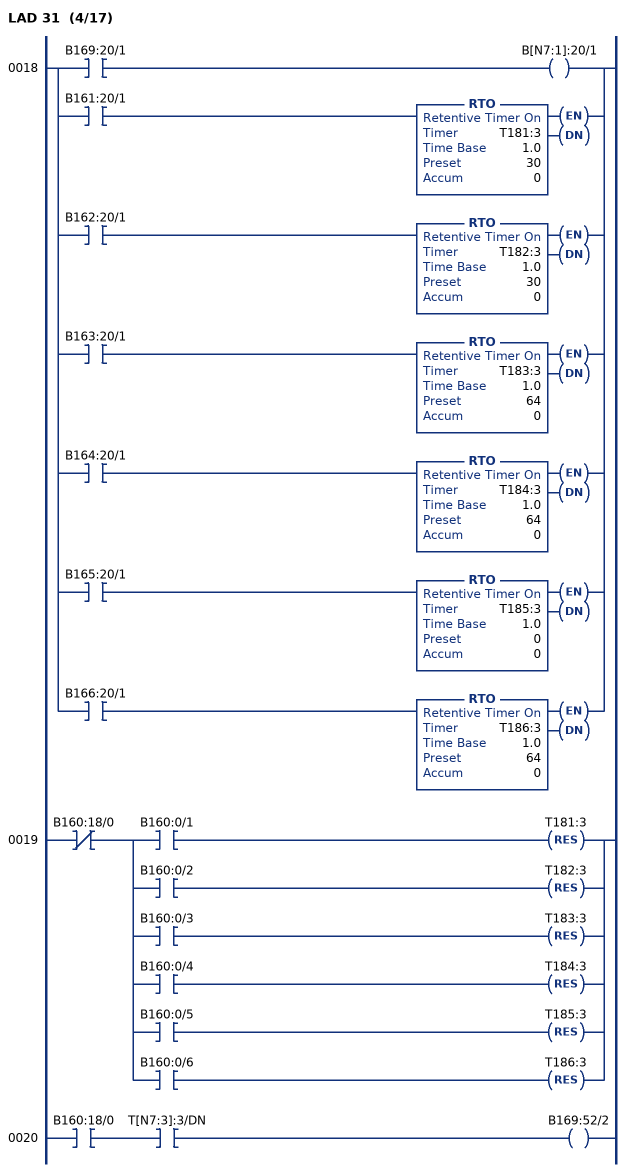
% Rung: 18 %
SOR BST XIC B169:20/1 OTE B[N7:1]:20/1 NXB XIC B161:20/1 RTO T181:3 1.0 30 0 NXB XIC B162:20/1 RTO T182:3 1.0 30 0 NXB XIC B163:20/1 RTO T183:3 1.0 64 0 NXB XIC B164:20/1 RTO T184:3 1.0 64 0 NXB XIC B165:20/1 RTO T185:3 1.0 0 0 NXB XIC B166:20/1 RTO T186:3 1.0 64 0 BND EOR
% Rung: 19 %
SOR XIO B160:18/0 BST XIC B160:0/1 RES T181:3 NXB XIC B160:0/2 RES T182:3 NXB XIC B160:0/3 RES T183:3 NXB XIC B160:0/4 RES T184:3 NXB XIC B160:0/5 RES T185:3 NXB XIC B160:0/6 RES T186:3 BND EOR
% Rung: 20 %
SOR XIC B160:18/0 XIC T[N7:3]:3/DN OTE B169:52/2 EOR

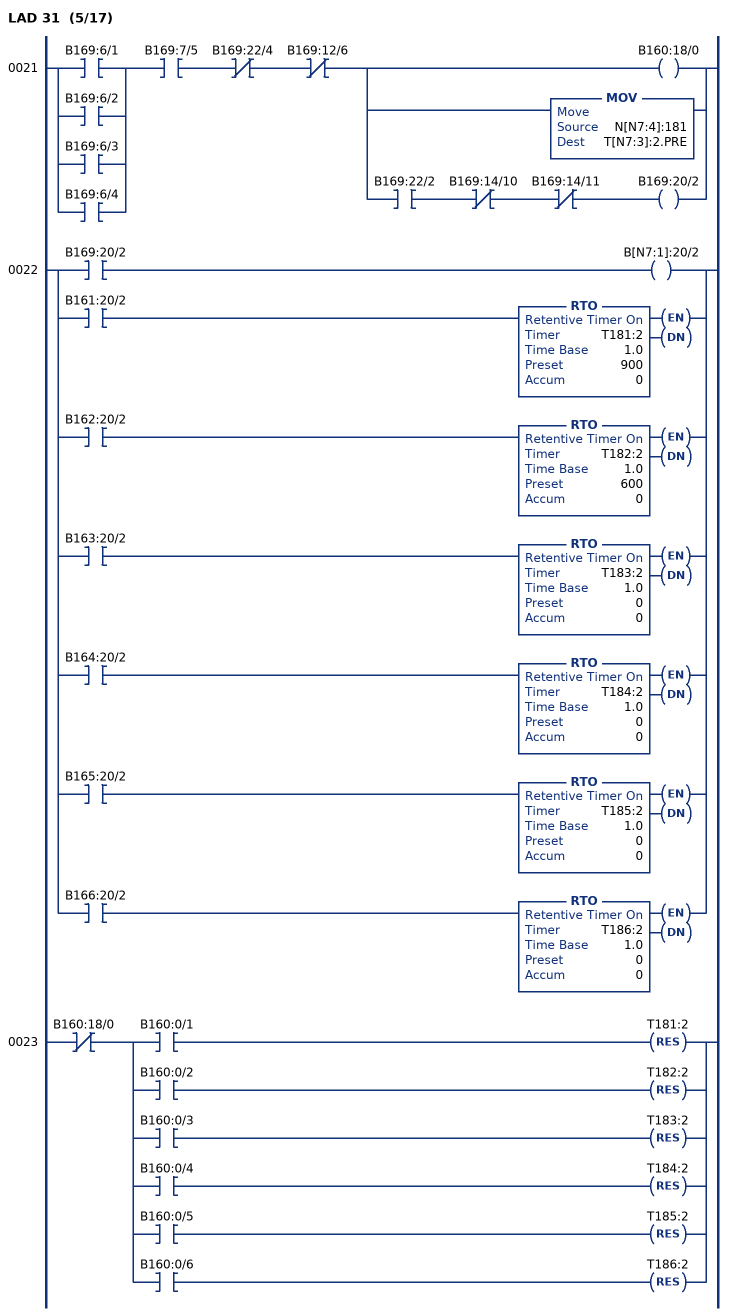
% Rung: 21 %
SOR BST XIC B169:6/1 NXB XIC B169:6/2 NXB XIC B169:6/3 NXB XIC B169:6/4 BND XIC B169:7/5 XIO B169:22/4 XIO B169:12/6 BST OTE B160:18/0 NXB MOV N[N7:4]:181 T[N7:3]:2.PRE NXB XIC B169:22/2 XIO B169:14/10 XIO B169:14/11 OTE B169:20/2 BND EOR
% Rung: 22 %
SOR BST XIC B169:20/2 OTE B[N7:1]:20/2 NXB XIC B161:20/2 RTO T181:2 1.0 900 0 NXB XIC B162:20/2 RTO T182:2 1.0 600 0 NXB XIC B163:20/2 RTO T183:2 1.0 0 0 NXB XIC B164:20/2 RTO T184:2 1.0 0 0 NXB XIC B165:20/2 RTO T185:2 1.0 0 0 NXB XIC B166:20/2 RTO T186:2 1.0 0 0 BND EOR
% Rung: 23 %
SOR XIO B160:18/0 BST XIC B160:0/1 RES T181:2 NXB XIC B160:0/2 RES T182:2 NXB XIC B160:0/3 RES T183:2 NXB XIC B160:0/4 RES T184:2 NXB XIC B160:0/5 RES T185:2 NXB XIC B160:0/6 RES T186:2 BND EOR

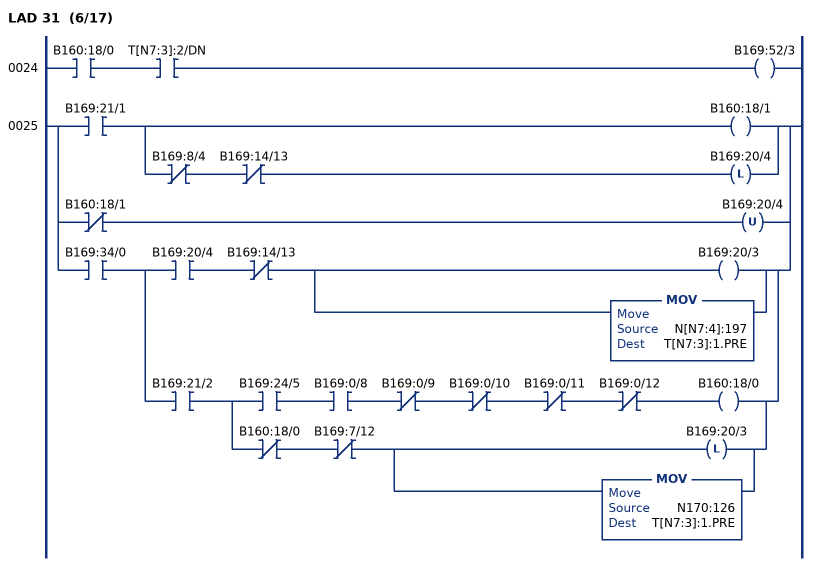
% Rung: 24 %
SOR XIC B160:18/0 XIC T[N7:3]:2/DN OTE B169:52/3 EOR
% Rung: 25 %
SOR BST XIC B169:21/1 BST OTE B160:18/1 NXB XIO B169:8/4 XIO B169:14/13 OTL B169:20/4 BND NXB XIO B160:18/1 OTU B169:20/4 NXB XIC B169:34/0 BST XIC B169:20/4 XIO B169:14/13 BST OTE B169:20/3 NXB MOV N[N7:4]:197 T[N7:3]:1.PRE BND NXB XIC B169:21/2 BST XIC B169:24/5 XIC B169:0/8 XIO B169:0/9 XIO B169:0/10 XIO B169:0/11 XIO B169:0/12 OTE B160:18/0 NXB XIO B160:18/0 XIO B169:7/12 BST OTL B169:20/3 NXB MOV N170:126 T[N7:3]:1.PRE BND BND BND BND EOR

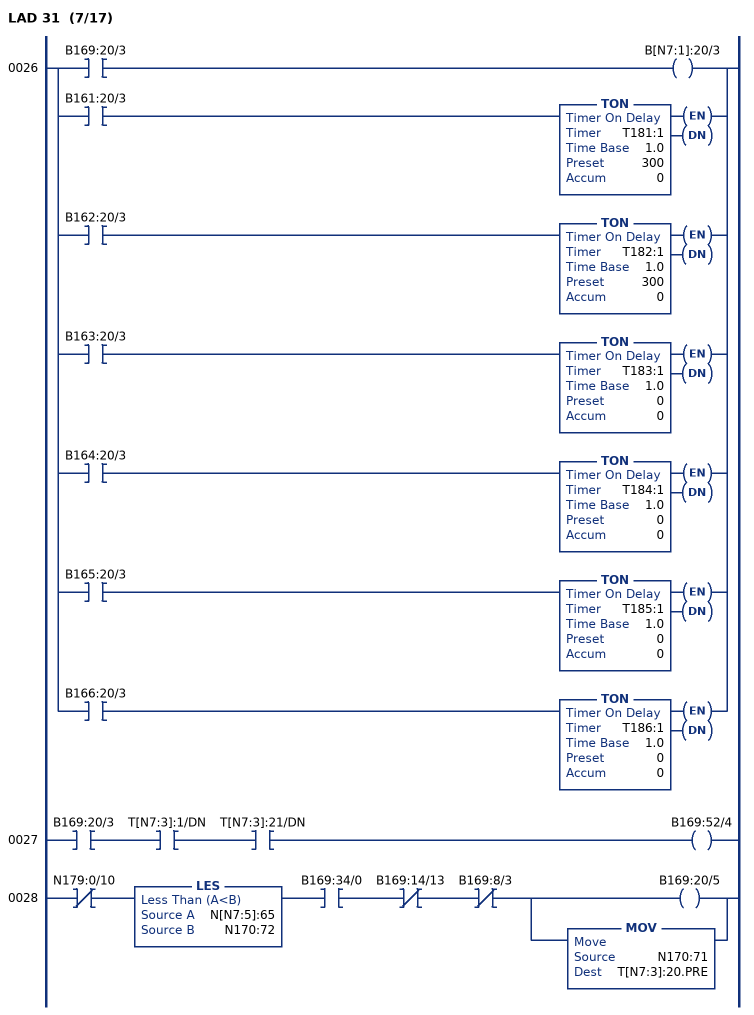
% Rung: 26 %
SOR BST XIC B169:20/3 OTE B[N7:1]:20/3 NXB XIC B161:20/3 TON T181:1 1.0 300 0 NXB XIC B162:20/3 TON T182:1 1.0 300 0 NXB XIC B163:20/3 TON T183:1 1.0 0 0 NXB XIC B164:20/3 TON T184:1 1.0 0 0 NXB XIC B165:20/3 TON T185:1 1.0 0 0 NXB XIC B166:20/3 TON T186:1 1.0 0 0 BND EOR
% Rung: 27 %
SOR XIC B169:20/3 XIC T[N7:3]:1/DN XIC T[N7:3]:21/DN OTE B169:52/4 EOR
% Rung: 28 %
SOR XIO N179:0/10 LES N[N7:5]:65 N170:72 XIC B169:34/0 XIO B169:14/13 XIO B169:8/3 BST OTE B169:20/5 NXB MOV N170:71 T[N7:3]:20.PRE BND EOR

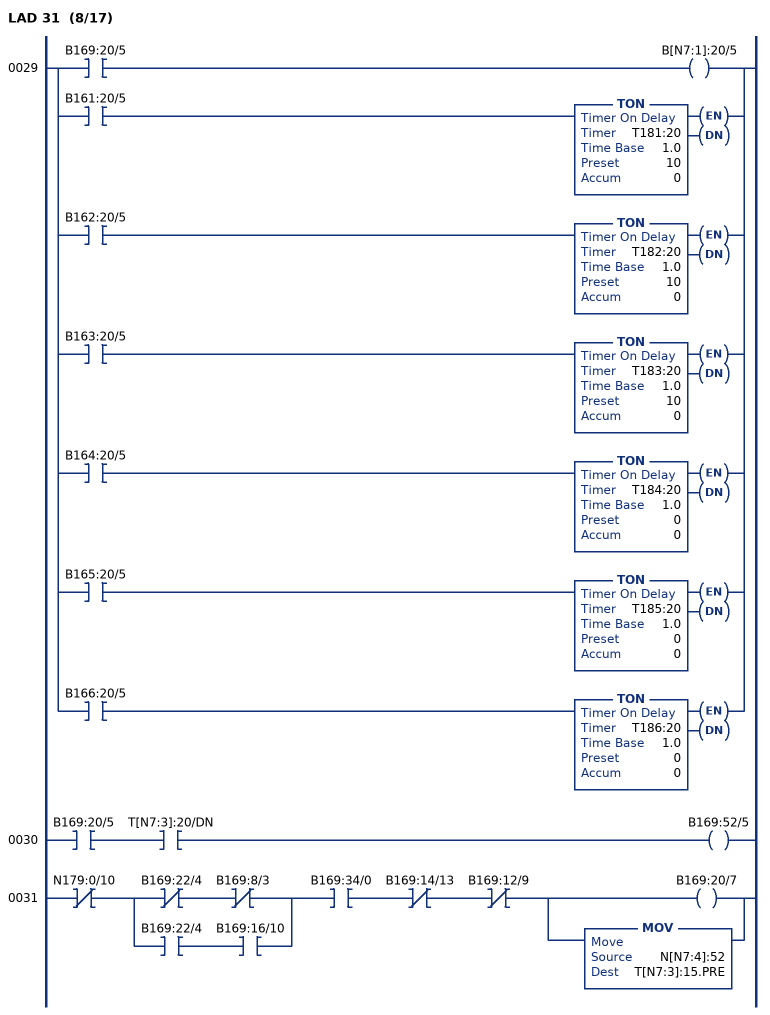
% Rung: 29 %
SOR BST XIC B169:20/5 OTE B[N7:1]:20/5 NXB XIC B161:20/5 TON T181:20 1.0 10 0 NXB XIC B162:20/5 TON T182:20 1.0 10 0 NXB XIC B163:20/5 TON T183:20 1.0 10 0 NXB XIC B164:20/5 TON T184:20 1.0 0 0 NXB XIC B165:20/5 TON T185:20 1.0 0 0 NXB XIC B166:20/5 TON T186:20 1.0 0 0 BND EOR
% Rung: 30 %
SOR XIC B169:20/5 XIC T[N7:3]:20/DN OTE B169:52/5 EOR
% Rung: 31 %
SOR XIO N179:0/10 BST XIO B169:22/4 XIO B169:8/3 NXB XIC B169:22/4 XIC B169:16/10 BND XIC B169:34/0 XIO B169:14/13 XIO B169:12/9 BST OTE B169:20/7 NXB MOV N[N7:4]:52 T[N7:3]:15.PRE BND EOR

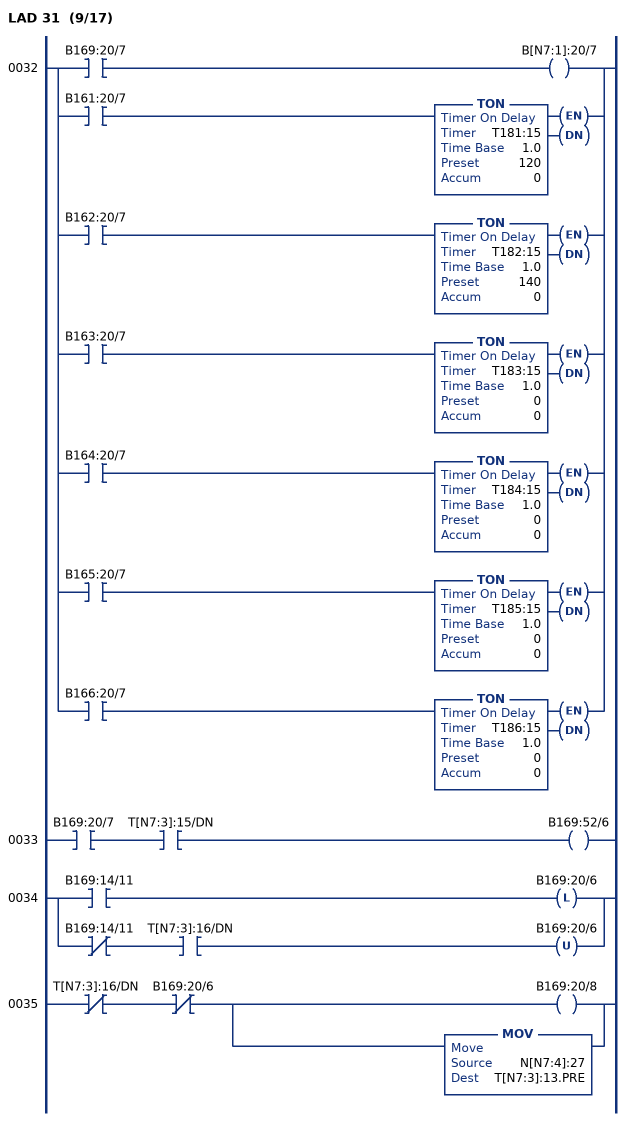
% Rung: 32 %
SOR BST XIC B169:20/7 OTE B[N7:1]:20/7 NXB XIC B161:20/7 TON T181:15 1.0 120 0 NXB XIC B162:20/7 TON T182:15 1.0 140 0 NXB XIC B163:20/7 TON T183:15 1.0 0 0 NXB XIC B164:20/7 TON T184:15 1.0 0 0 NXB XIC B165:20/7 TON T185:15 1.0 0 0 NXB XIC B166:20/7 TON T186:15 1.0 0 0 BND EOR
% Rung: 33 %
SOR XIC B169:20/7 XIC T[N7:3]:15/DN OTE B169:52/6 EOR
% Rung: 34 %
SOR BST XIC B169:14/11 OTL B169:20/6 NXB XIO B169:14/11 XIC T[N7:3]:16/DN OTU B169:20/6 BND EOR
% Rung: 35 %
SOR XIO T[N7:3]:16/DN XIO B169:20/6 BST OTE B169:20/8 NXB MOV N[N7:4]:27 T[N7:3]:13.PRE BND EOR

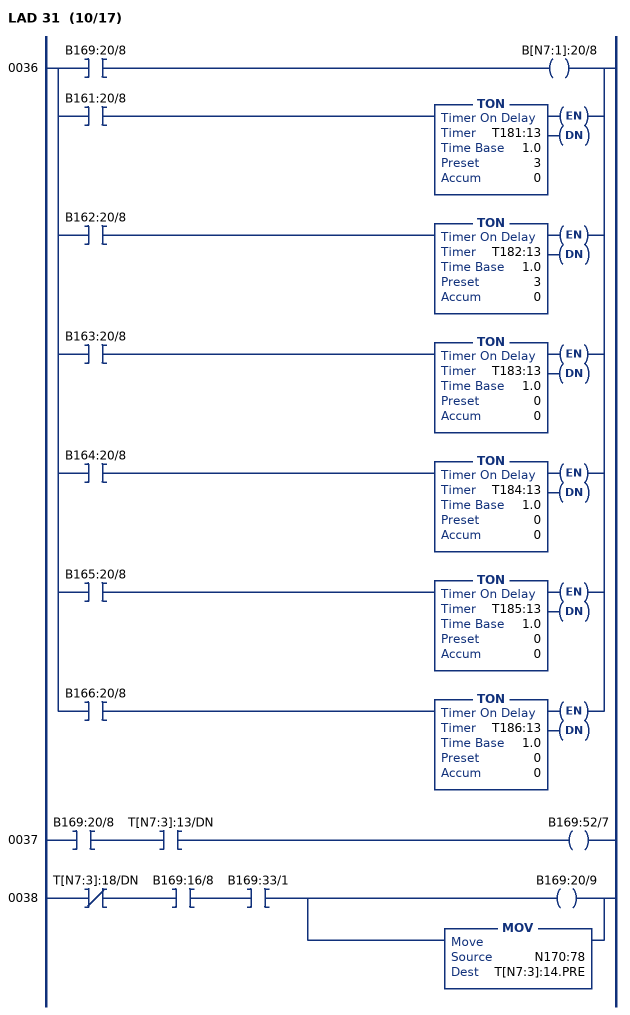
% Rung: 36 %
SOR BST XIC B169:20/8 OTE B[N7:1]:20/8 NXB XIC B161:20/8 TON T181:13 1.0 3 0 NXB XIC B162:20/8 TON T182:13 1.0 3 0 NXB XIC B163:20/8 TON T183:13 1.0 0 0 NXB XIC B164:20/8 TON T184:13 1.0 0 0 NXB XIC B165:20/8 TON T185:13 1.0 0 0 NXB XIC B166:20/8 TON T186:13 1.0 0 0 BND EOR
% Rung: 37 %
SOR XIC B169:20/8 XIC T[N7:3]:13/DN OTE B169:52/7 EOR
% Rung: 38 %
SOR XIO T[N7:3]:18/DN XIC B169:16/8 XIC B169:33/1 BST OTE B169:20/9 NXB MOV N170:78 T[N7:3]:14.PRE BND EOR

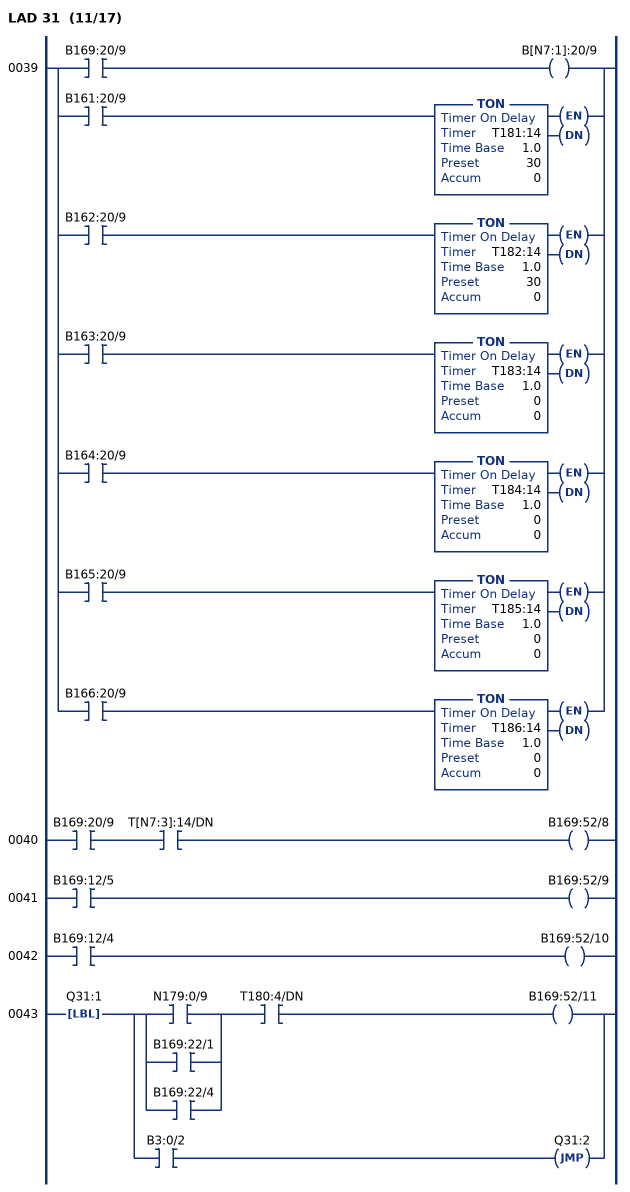
% Rung: 39 %
SOR BST XIC B169:20/9 OTE B[N7:1]:20/9 NXB XIC B161:20/9 TON T181:14 1.0 30 0 NXB XIC B162:20/9 TON T182:14 1.0 30 0 NXB XIC B163:20/9 TON T183:14 1.0 0 0 NXB XIC B164:20/9 TON T184:14 1.0 0 0 NXB XIC B165:20/9 TON T185:14 1.0 0 0 NXB XIC B166:20/9 TON T186:14 1.0 0 0 BND EOR
% Rung: 40 %
SOR XIC B169:20/9 XIC T[N7:3]:14/DN OTE B169:52/8 EOR
% Rung: 41 %
SOR XIC B169:12/5 OTE B169:52/9 EOR
% Rung: 42 %
SOR XIC B169:12/4 OTE B169:52/10 EOR
% Rung: 43 %
SOR LBL Q31:1 BST BST XIC N179:0/9 NXB XIC B169:22/1 NXB XIC B169:22/4 BND XIC T180:4/DN OTE B169:52/11 NXB XIC B3:0/2 JMP Q31:2 BND EOR

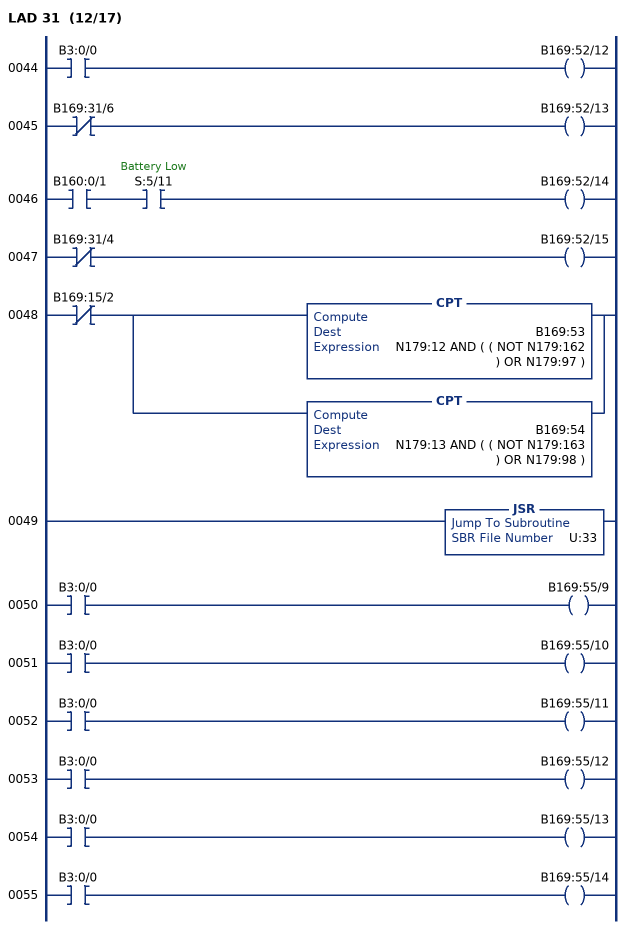
% Rung: 44 %
SOR XIC B3:0/0 OTE B169:52/12 EOR
% Rung: 45 %
SOR XIO B169:31/6 OTE B169:52/13 EOR
% Rung: 46 %
SOR XIC B160:0/1 XIC S:5/11 OTE B169:52/14 EOR
%   S:5/11  "Battery Low" %
% Rung: 47 %
SOR XIO B169:31/4 OTE B169:52/15 EOR
% Rung: 48 %
SOR XIO B169:15/2 BST CPT B169:53 " N179:12 AND ( ( NOT N179:162 ) OR N179:97 ) " NXB CPT B169:54 " N179:13 AND ( ( NOT N179:163 ) OR N179:98 ) " BND EOR
% Rung: 49 %
SOR JSR U:33 EOR
% Rung: 50 %
SOR XIC B3:0/0 OTE B169:55/9 EOR
% Rung: 51 %
SOR XIC B3:0/0 OTE B169:55/10 EOR
% Rung: 52 %
SOR XIC B3:0/0 OTE B169:55/11 EOR
% Rung: 53 %
SOR XIC B3:0/0 OTE B169:55/12 EOR
% Rung: 54 %
SOR XIC B3:0/0 OTE B169:55/13 EOR
% Rung: 55 %
SOR XIC B3:0/0 OTE B169:55/14 EOR

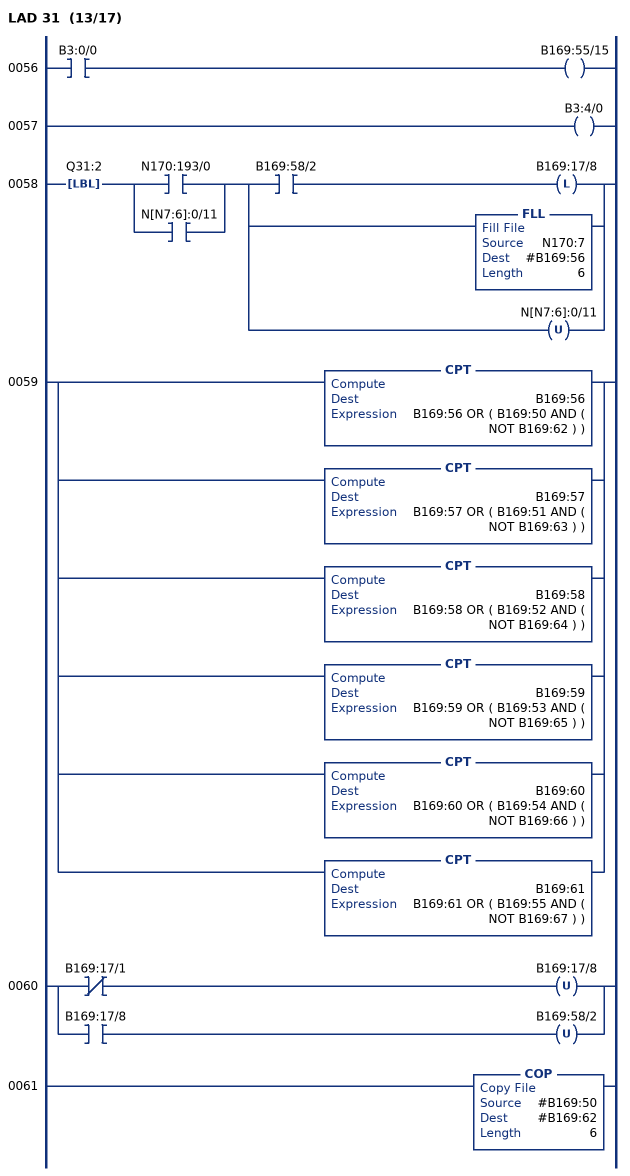
% Rung: 56 %
SOR XIC B3:0/0 OTE B169:55/15 EOR
% Rung: 57 %
SOR OTE B3:4/0 EOR
% Rung: 58 %
SOR LBL Q31:2 BST XIC N170:193/0 NXB XIC N[N7:6]:0/11 BND BST XIC B169:58/2 OTL B169:17/8 NXB FLL N170:7 #B169:56 6 NXB OTU N[N7:6]:0/11 BND EOR
% Rung: 59 %
SOR BST CPT B169:56 " B169:56 OR ( B169:50 AND ( NOT B169:62 ) ) " NXB CPT B169:57 " B169:57 OR ( B169:51 AND ( NOT B169:63 ) ) " NXB CPT B169:58 " B169:58 OR ( B169:52 AND ( NOT B169:64 ) ) " NXB CPT B169:59 " B169:59 OR ( B169:53 AND ( NOT B169:65 ) ) " NXB CPT B169:60 " B169:60 OR ( B169:54 AND ( NOT B169:66 ) ) " NXB CPT B169:61 " B169:61 OR ( B169:55 AND ( NOT B169:67 ) ) " BND EOR
% Rung: 60 %
SOR BST XIO B169:17/1 OTU B169:17/8 NXB XIC B169:17/8 OTU B169:58/2 BND EOR
% Rung: 61 %
SOR COP #B169:50 #B169:62 6 EOR

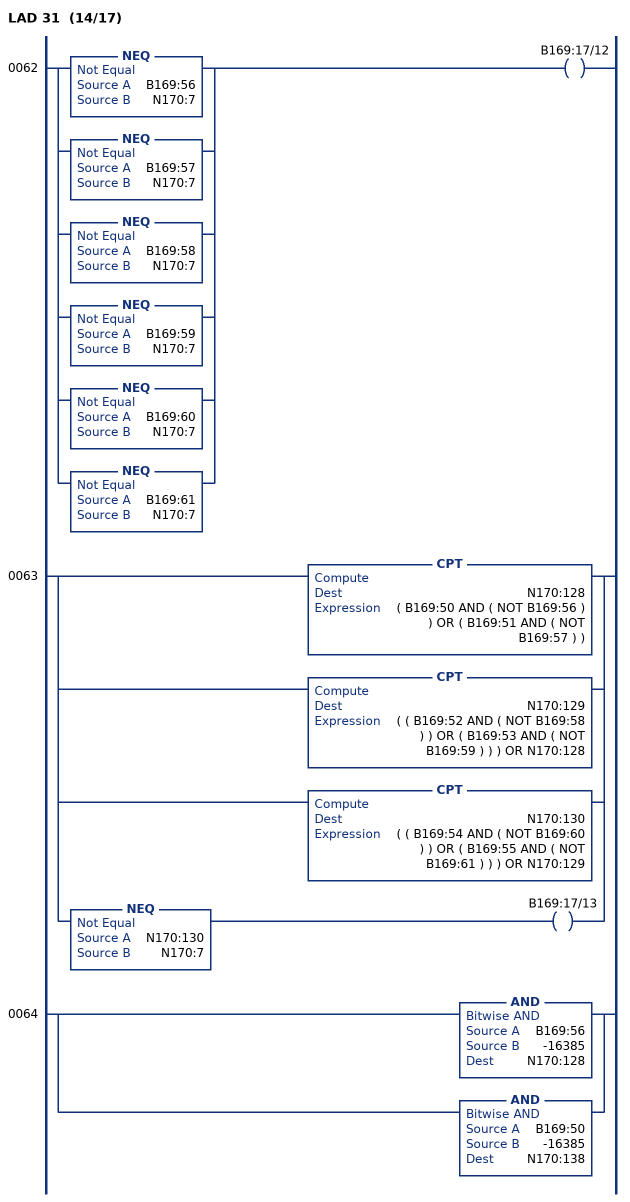
% Rung: 62 %
SOR BST NEQ B169:56 N170:7 NXB NEQ B169:57 N170:7 NXB NEQ B169:58 N170:7 NXB NEQ B169:59 N170:7 NXB NEQ B169:60 N170:7 NXB NEQ B169:61 N170:7 BND OTE B169:17/12 EOR
% Rung: 63 %
SOR BST CPT N170:128 " ( B169:50 AND ( NOT B169:56 ) ) OR ( B169:51 AND ( NOT B169:57 ) ) " NXB CPT N170:129 " ( ( B169:52 AND ( NOT B169:58 ) ) OR ( B169:53 AND ( NOT B169:59 ) ) ) OR N170:128 " NXB CPT N170:130 " ( ( B169:54 AND ( NOT B169:60 ) ) OR ( B169:55 AND ( NOT B169:61 ) ) ) OR N170:129 " NXB NEQ N170:130 N170:7 OTE B169:17/13 BND EOR
% Rung: 64 %
SOR BST AND B169:56 -16385 N170:128 NXB AND B169:50 -16385 N170:138 BND EOR

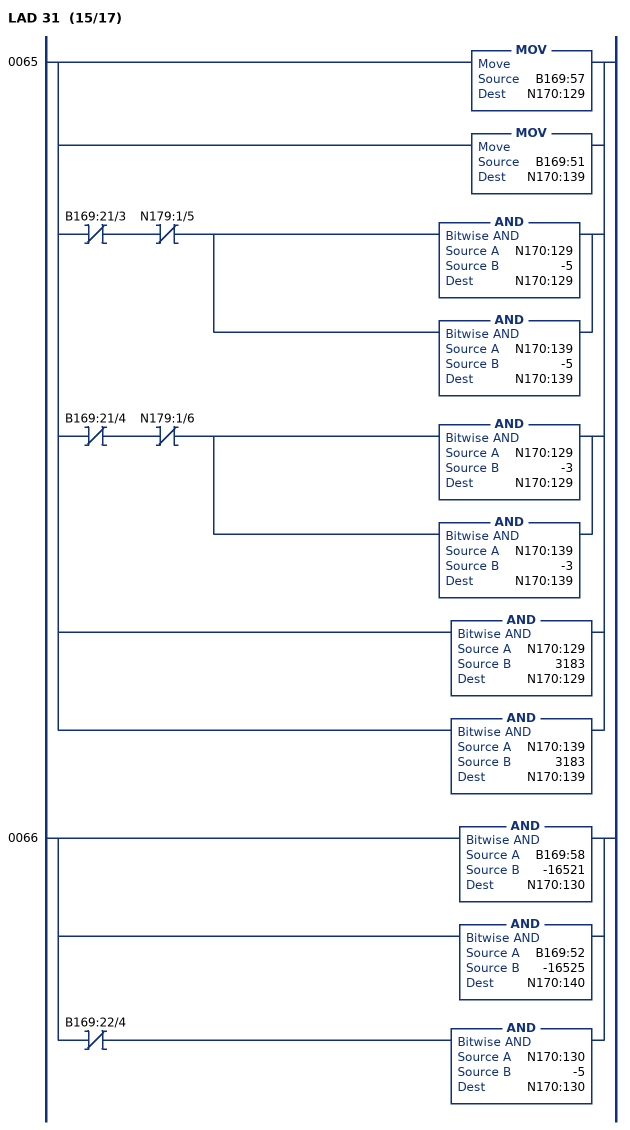
% Rung: 65 %
SOR BST MOV B169:57 N170:129 NXB MOV B169:51 N170:139 NXB XIO B169:21/3 XIO N179:1/5 BST AND N170:129 -5 N170:129 NXB AND N170:139 -5 N170:139 BND NXB XIO B169:21/4 XIO N179:1/6 BST AND N170:129 -3 N170:129 NXB AND N170:139 -3 N170:139 BND NXB AND N170:129 3183 N170:129 NXB AND N170:139 3183 N170:139 BND EOR
% Rung: 66 %
SOR BST AND B169:58 -16521 N170:130 NXB AND B169:52 -16525 N170:140 NXB XIO B169:22/4 AND N170:130 -5 N170:130 BND EOR

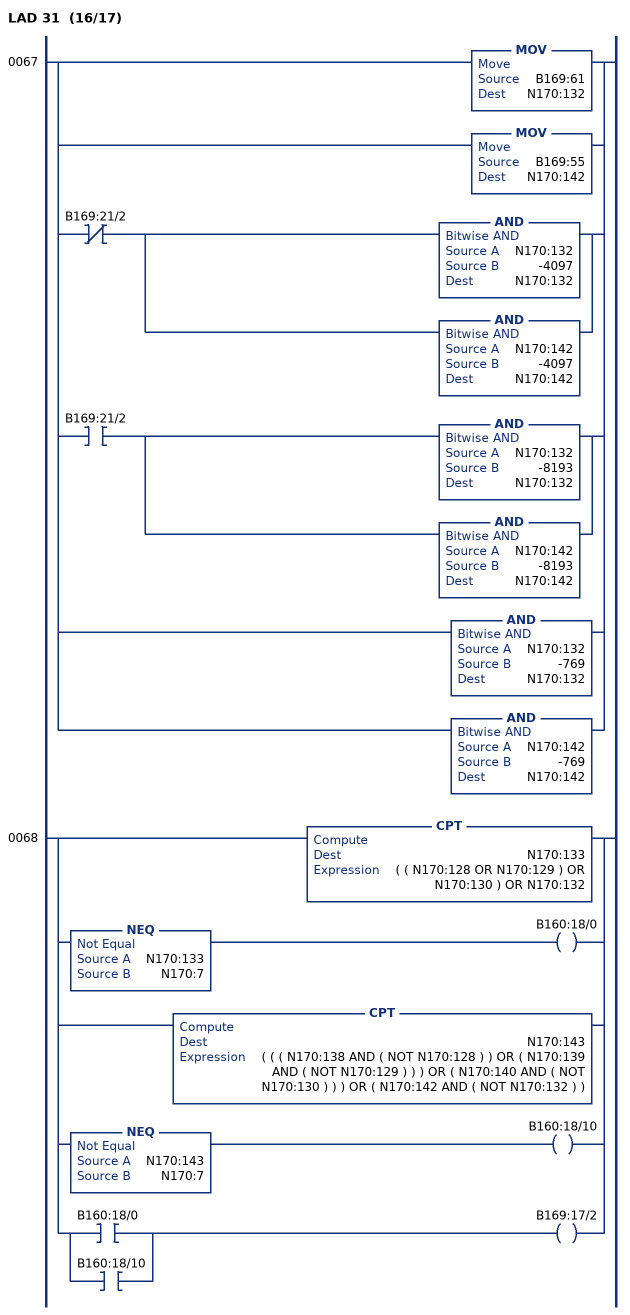
% Rung: 67 %
SOR BST MOV B169:61 N170:132 NXB MOV B169:55 N170:142 NXB XIO B169:21/2 BST AND N170:132 -4097 N170:132 NXB AND N170:142 -4097 N170:142 BND NXB XIC B169:21/2 BST AND N170:132 -8193 N170:132 NXB AND N170:142 -8193 N170:142 BND NXB AND N170:132 -769 N170:132 NXB AND N170:142 -769 N170:142 BND EOR
% Rung: 68 %
SOR BST CPT N170:133 " ( ( N170:128 OR N170:129 ) OR N170:130 ) OR N170:132 " NXB NEQ N170:133 N170:7 OTE B160:18/0 NXB CPT N170:143 " ( ( ( N170:138 AND ( NOT N170:128 ) ) OR ( N170:139 AND ( NOT N170:129 ) ) ) OR ( N170:140 AND ( NOT N170:130 ) ) ) OR ( N170:142 AND ( NOT N170:132 ) ) " NXB NEQ N170:143 N170:7 OTE B160:18/10 NXB BST XIC B160:18/0 NXB XIC B160:18/10 BND OTE B169:17/2 BND EOR

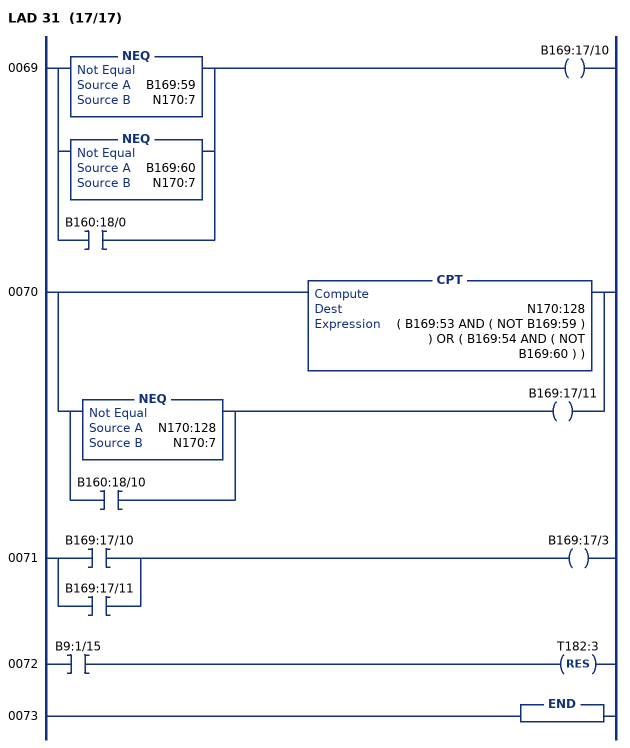
% Rung: 69 %
SOR BST NEQ B169:59 N170:7 NXB NEQ B169:60 N170:7 NXB XIC B160:18/0 BND OTE B169:17/10 EOR
% Rung: 70 %
SOR BST CPT N170:128 " ( B169:53 AND ( NOT B169:59 ) ) OR ( B169:54 AND ( NOT B169:60 ) ) " NXB BST NEQ N170:128 N170:7 NXB XIC B160:18/10 BND OTE B169:17/11 BND EOR
% Rung: 71 %
SOR BST XIC B169:17/10 NXB XIC B169:17/11 BND OTE B169:17/3 EOR
% Rung: 72 %
SOR XIC B9:1/15 RES T182:3 EOR
% Rung: 73 %
SOR END EOR

LADDER 32
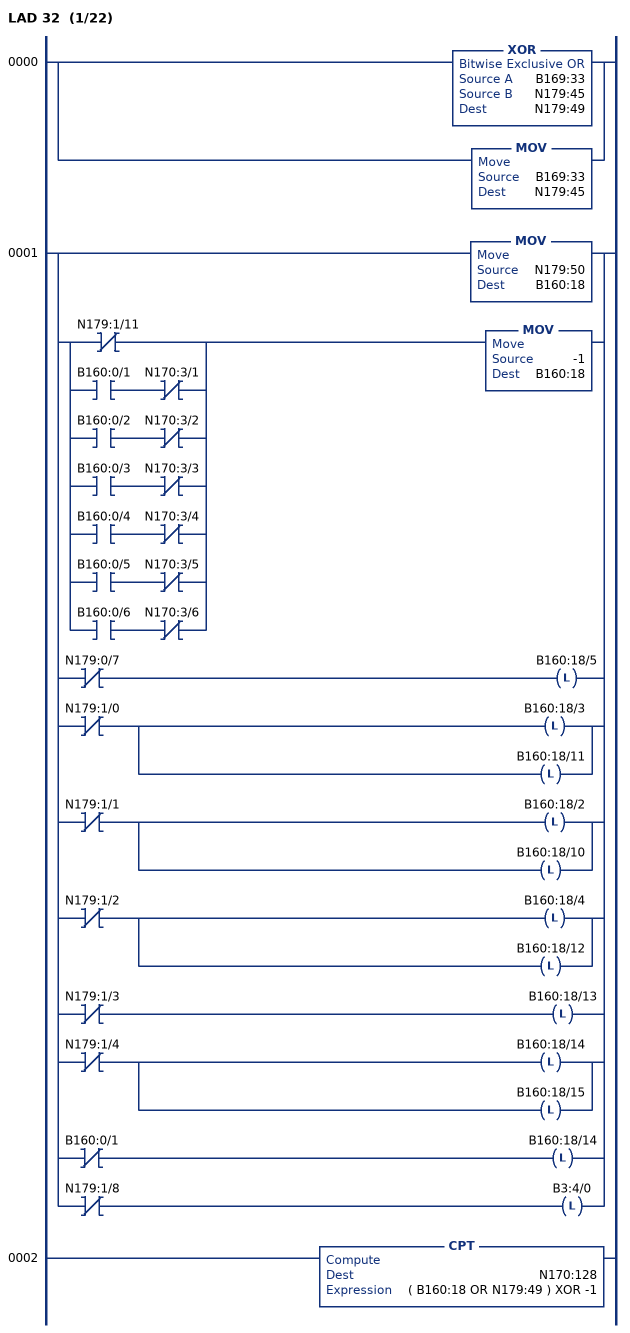
% Rung: 0 %
SOR BST XOR B169:33 N179:45 N179:49 NXB MOV B169:33 N179:45 BND EOR
% Rung: 1 %
SOR BST MOV N179:50 B160:18 NXB BST XIO N179:1/11 NXB XIC B160:0/1 XIO N170:3/1 NXB XIC B160:0/2 XIO N170:3/2 NXB XIC B160:0/3 XIO N170:3/3 NXB XIC B160:0/4 XIO N170:3/4 NXB XIC B160:0/5 XIO N170:3/5 NXB XIC B160:0/6 XIO N170:3/6 BND MOV -1 B160:18 NXB XIO N179:0/7 OTL B160:18/5 NXB XIO N179:1/0 BST OTL B160:18/3 NXB OTL B160:18/11 BND NXB XIO N179:1/1 BST OTL B160:18/2 NXB OTL B160:18/10 BND NXB XIO N179:1/2 BST OTL B160:18/4 NXB OTL B160:18/12 BND NXB XIO N179:1/3 OTL B160:18/13 NXB BST XIO N179:1/4 BST OTL B160:18/14 NXB OTL B160:18/15 BND NXB XIO B160:0/1 OTL B160:18/14 BND NXB XIO N179:1/8 OTL B3:4/0 BND EOR
% Rung: 2 %
SOR CPT N170:128 " ( B160:18 OR N179:49 ) XOR -1 " EOR

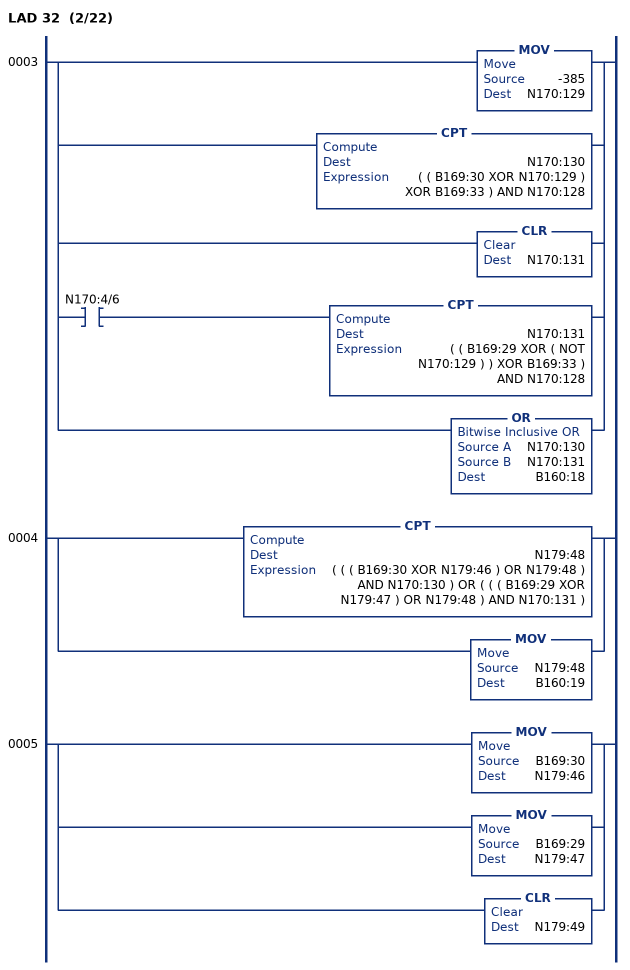
% Rung: 3 %
SOR BST MOV -385 N170:129 NXB CPT N170:130 " ( ( B169:30 XOR N170:129 ) XOR B169:33 ) AND N170:128 " NXB CLR N170:131 NXB XIC N170:4/6 CPT N170:131 " ( ( B169:29 XOR ( NOT N170:129 ) ) XOR B169:33 ) AND N170:128 " NXB OR N170:130 N170:131 B160:18 BND EOR
% Rung: 4 %
SOR BST CPT N179:48 " ( ( ( B169:30 XOR N179:46 ) OR N179:48 ) AND N170:130 ) OR ( ( ( B169:29 XOR N179:47 ) OR N179:48 ) AND N170:131 ) " NXB MOV N179:48 B160:19 BND EOR
% Rung: 5 %
SOR BST MOV B169:30 N179:46 NXB MOV B169:29 N179:47 NXB CLR N179:49 BND EOR

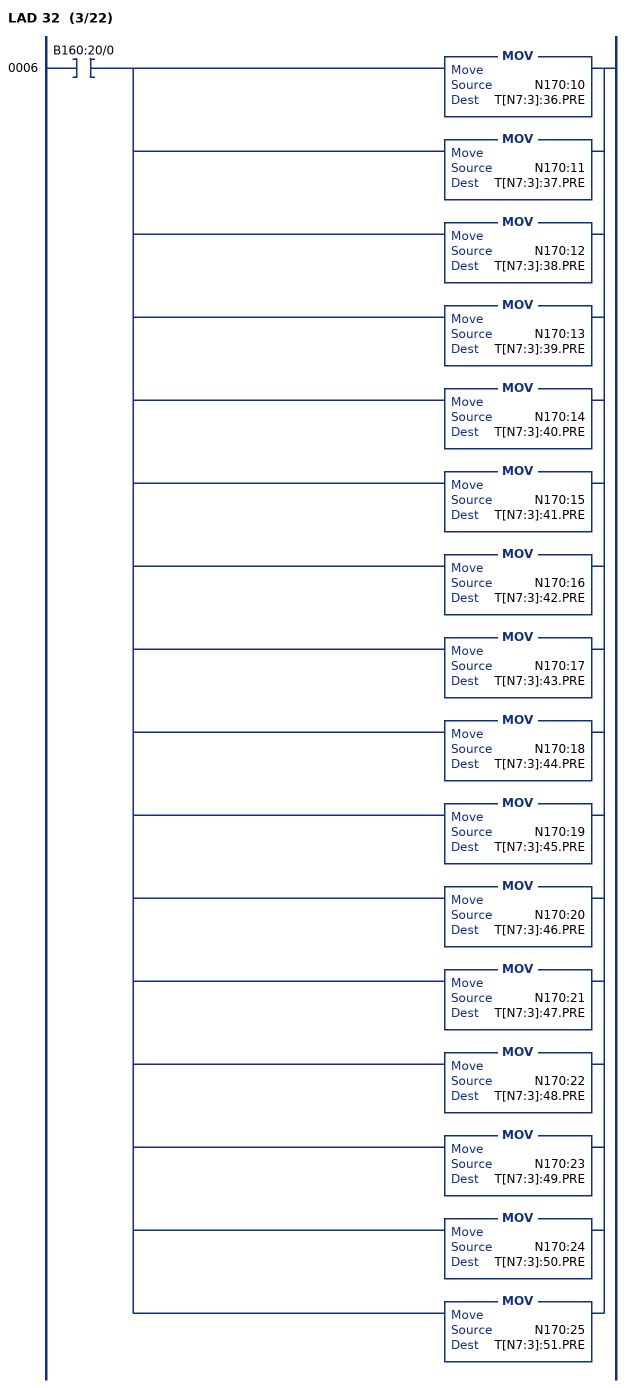
% Rung: 6 %
SOR XIC B160:20/0 BST MOV N170:10 T[N7:3]:36.PRE NXB MOV N170:11 T[N7:3]:37.PRE NXB MOV N170:12 T[N7:3]:38.PRE NXB MOV N170:13 T[N7:3]:39.PRE NXB MOV N170:14 T[N7:3]:40.PRE NXB MOV N170:15 T[N7:3]:41.PRE NXB MOV N170:16 T[N7:3]:42.PRE NXB MOV N170:17 T[N7:3]:43.PRE NXB MOV N170:18 T[N7:3]:44.PRE NXB MOV N170:19 T[N7:3]:45.PRE NXB MOV N170:20 T[N7:3]:46.PRE NXB MOV N170:21 T[N7:3]:47.PRE NXB MOV N170:22 T[N7:3]:48.PRE NXB MOV N170:23 T[N7:3]:49.PRE NXB MOV N170:24 T[N7:3]:50.PRE NXB MOV N170:25 T[N7:3]:51.PRE BND EOR

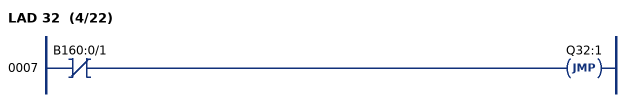
% Rung: 7 %
SOR XIO B160:0/1 JMP Q32:1 EOR

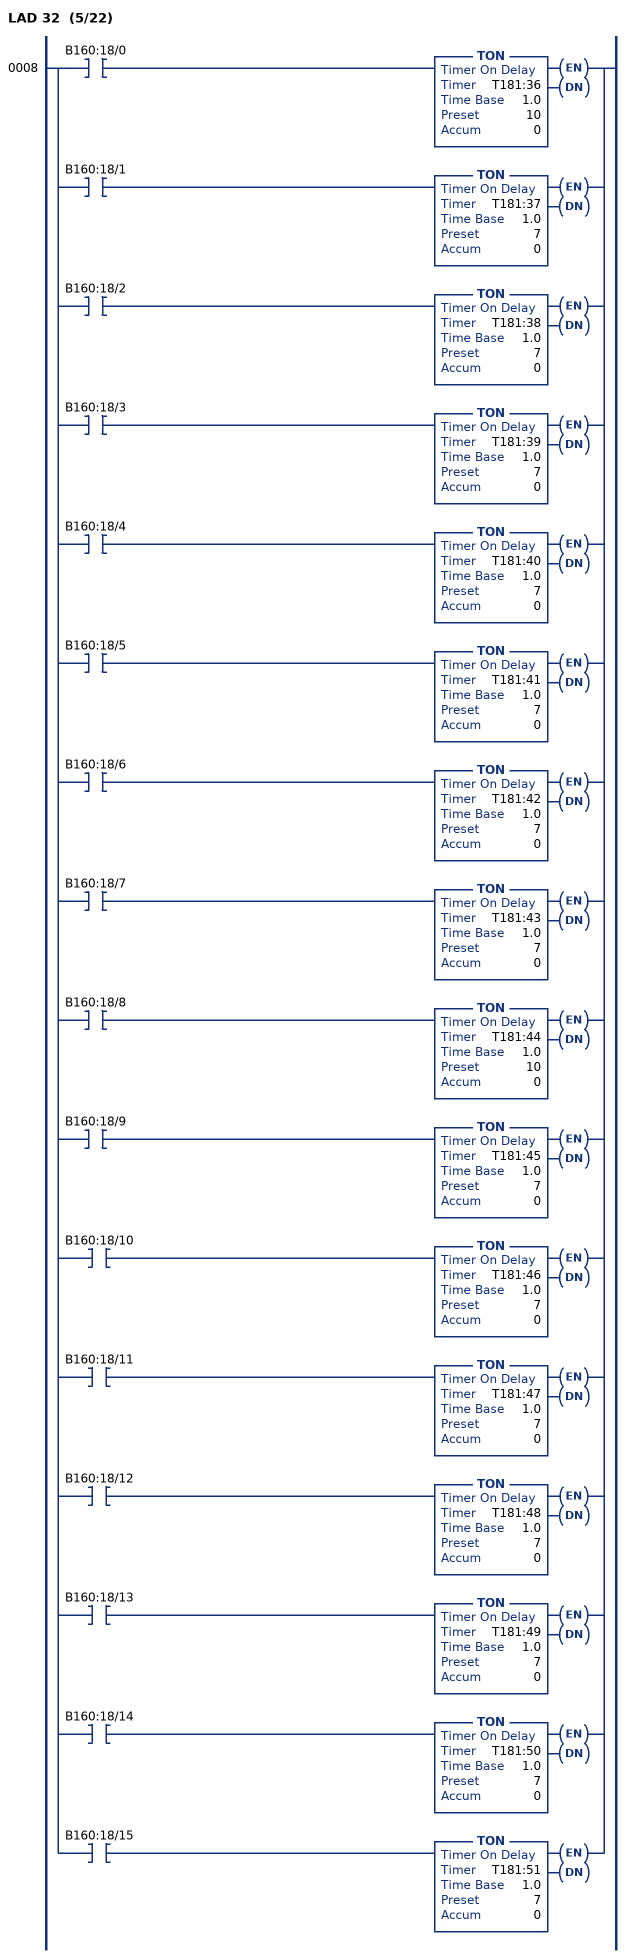
% Rung: 8 %
SOR BST XIC B160:18/0 TON T181:36 1.0 10 0 NXB XIC B160:18/1 TON T181:37 1.0 7 0 NXB XIC B160:18/2 TON T181:38 1.0 7 0 NXB XIC B160:18/3 TON T181:39 1.0 7 0 NXB XIC B160:18/4 TON T181:40 1.0 7 0 NXB XIC B160:18/5 TON T181:41 1.0 7 0 NXB XIC B160:18/6 TON T181:42 1.0 7 0 NXB XIC B160:18/7 TON T181:43 1.0 7 0 NXB XIC B160:18/8 TON T181:44 1.0 10 0 NXB XIC B160:18/9 TON T181:45 1.0 7 0 NXB XIC B160:18/10 TON T181:46 1.0 7 0 NXB XIC B160:18/11 TON T181:47 1.0 7 0 NXB XIC B160:18/12 TON T181:48 1.0 7 0 NXB XIC B160:18/13 TON T181:49 1.0 7 0 NXB XIC B160:18/14 TON T181:50 1.0 7 0 NXB XIC B160:18/15 TON T181:51 1.0 7 0 BND EOR

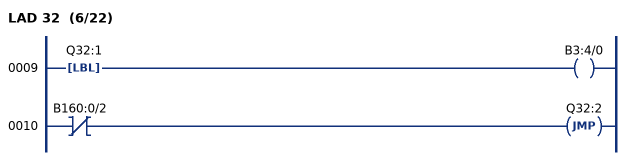
% Rung: 9 %
SOR LBL Q32:1 OTE B3:4/0 EOR
% Rung: 10 %
SOR XIO B160:0/2 JMP Q32:2 EOR

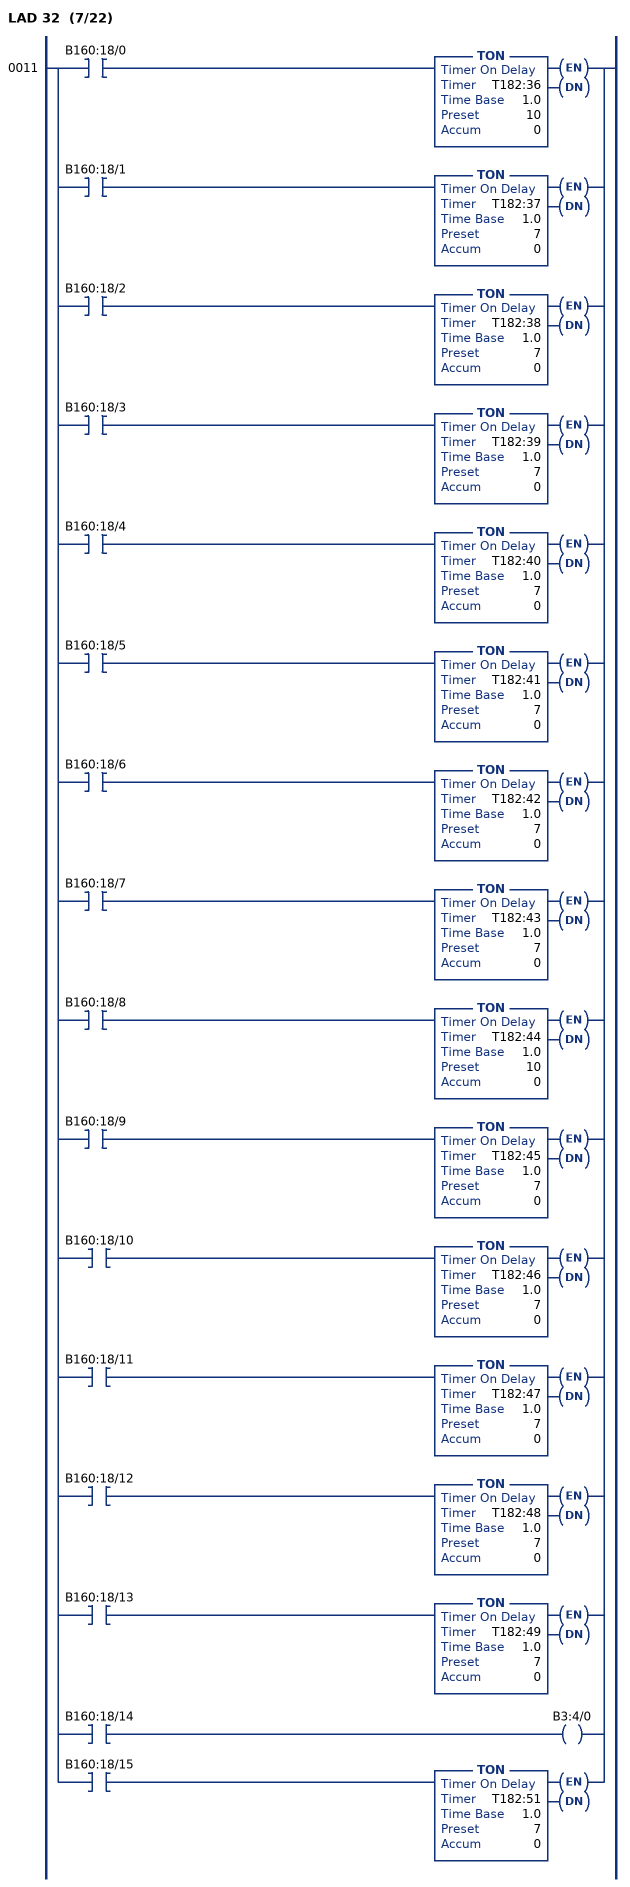
% Rung: 11 %
SOR BST XIC B160:18/0 TON T182:36 1.0 10 0 NXB XIC B160:18/1 TON T182:37 1.0 7 0 NXB XIC B160:18/2 TON T182:38 1.0 7 0 NXB XIC B160:18/3 TON T182:39 1.0 7 0 NXB XIC B160:18/4 TON T182:40 1.0 7 0 NXB XIC B160:18/5 TON T182:41 1.0 7 0 NXB XIC B160:18/6 TON T182:42 1.0 7 0 NXB XIC B160:18/7 TON T182:43 1.0 7 0 NXB XIC B160:18/8 TON T182:44 1.0 10 0 NXB XIC B160:18/9 TON T182:45 1.0 7 0 NXB XIC B160:18/10 TON T182:46 1.0 7 0 NXB XIC B160:18/11 TON T182:47 1.0 7 0 NXB XIC B160:18/12 TON T182:48 1.0 7 0 NXB XIC B160:18/13 TON T182:49 1.0 7 0 NXB XIC B160:18/14 OTE B3:4/0 NXB XIC B160:18/15 TON T182:51 1.0 7 0 BND EOR

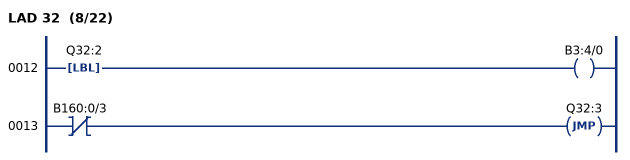
% Rung: 12 %
SOR LBL Q32:2 OTE B3:4/0 EOR
% Rung: 13 %
SOR XIO B160:0/3 JMP Q32:3 EOR

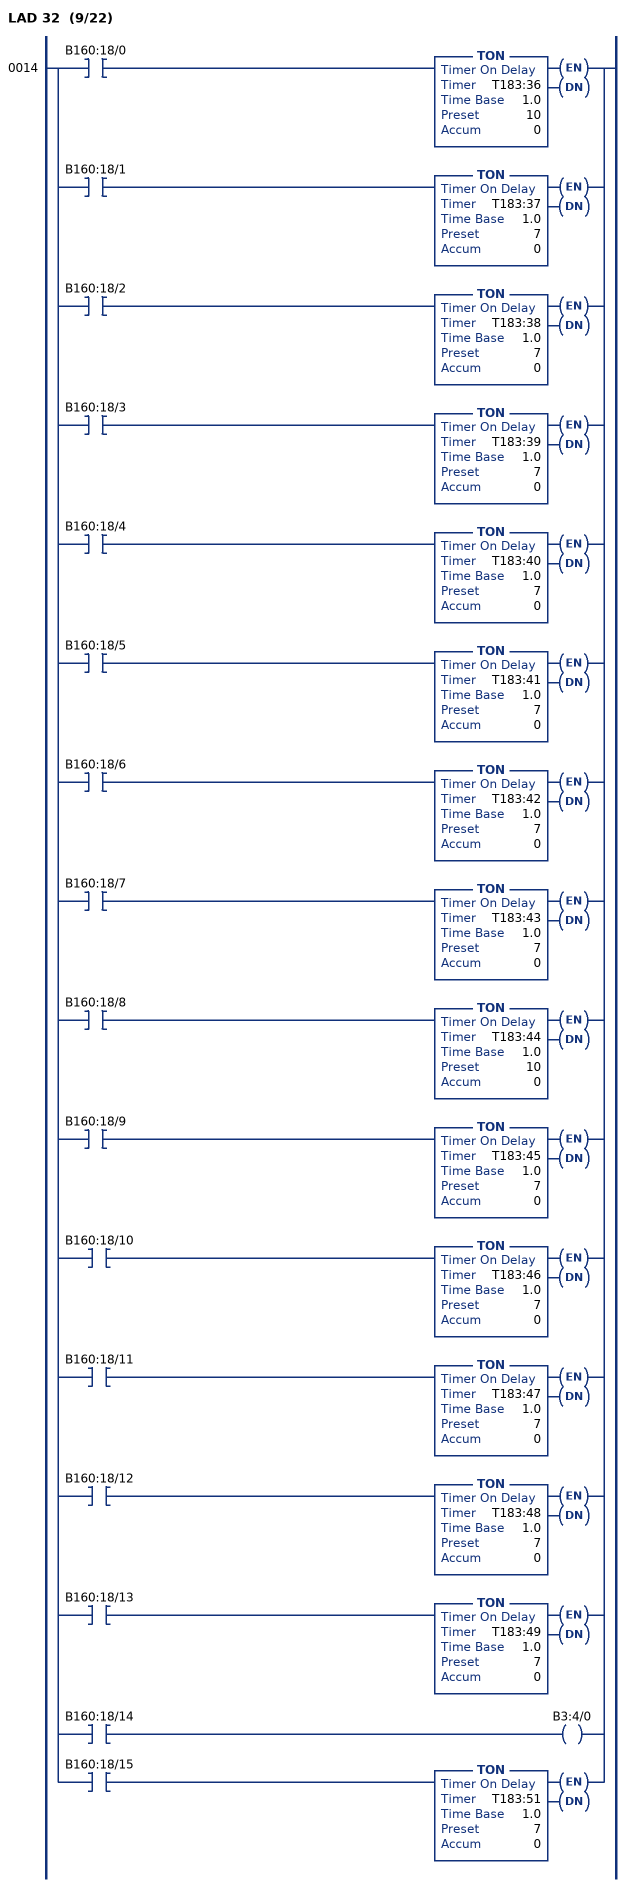
% Rung: 14 %
SOR BST XIC B160:18/0 TON T183:36 1.0 10 0 NXB XIC B160:18/1 TON T183:37 1.0 7 0 NXB XIC B160:18/2 TON T183:38 1.0 7 0 NXB XIC B160:18/3 TON T183:39 1.0 7 0 NXB XIC B160:18/4 TON T183:40 1.0 7 0 NXB XIC B160:18/5 TON T183:41 1.0 7 0 NXB XIC B160:18/6 TON T183:42 1.0 7 0 NXB XIC B160:18/7 TON T183:43 1.0 7 0 NXB XIC B160:18/8 TON T183:44 1.0 10 0 NXB XIC B160:18/9 TON T183:45 1.0 7 0 NXB XIC B160:18/10 TON T183:46 1.0 7 0 NXB XIC B160:18/11 TON T183:47 1.0 7 0 NXB XIC B160:18/12 TON T183:48 1.0 7 0 NXB XIC B160:18/13 TON T183:49 1.0 7 0 NXB XIC B160:18/14 OTE B3:4/0 NXB XIC B160:18/15 TON T183:51 1.0 7 0 BND EOR

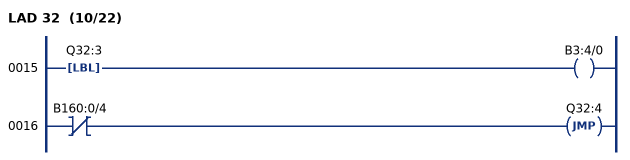
% Rung: 15 %
SOR LBL Q32:3 OTE B3:4/0 EOR
% Rung: 16 %
SOR XIO B160:0/4 JMP Q32:4 EOR

